Universal Robots PolyScope program: testy.urp

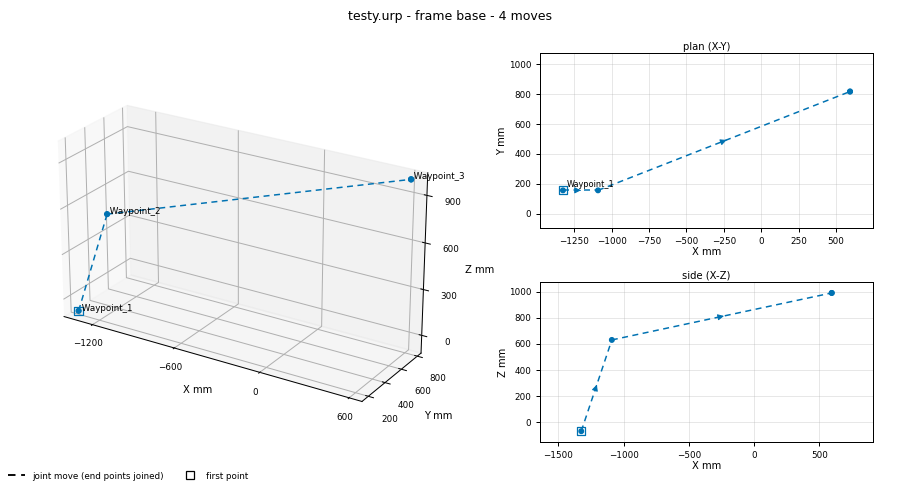
[picture p0: tool path of testy.urp in frame base, 4 of 4 moves have a stored position in this frame; points joined in program order, loops and branches not executed]
Program testy (installation=default directory=/programs createdIn=5.21.3 lastSavedIn=5.21.3 robotSerialNumber=20246801938)
Calibrated DH parameters: a=[-0.000071, -0.790281, -0.600694, 0.000061, -0.000039, 0]; d=[0.236272, 604.465945, 132.116513, -736.382239, 0.159268, 0.154005]; alpha=[1.570254, -0.000567, 0.000559, 1.571709, -1.56999, 0]; deltaTheta=[0, -0.409357, 7.293326, -0.600784, -0.000001, -0.000001]
InitVariablesNode
Robot Program (runOnlyOnce=false)
  'weld angle'
  MoveJ speed 60 deg/s, acceleration 80 deg/s^2 (useActiveTCP=true optimoveEnabled=false optiMoveSpeed=0.3 optiMoveAcceleration=0.09) feature=Base
    Waypoint Waypoint_1: TCP in base x=-1325.071 y=156.59 z=-68.113 mm, rx=-1.7149 ry=0.7798 rz=1.7149 rad; joints [-6.175, -45.066, 109.192, 205.921, -90.048, 42.74] deg; TCP offset x=-11.7 y=-328 z=105 mm, rx=1.2092 ry=-1.2092 rz=1.2092 rad
    Waypoint Waypoint_2: TCP in base x=-1090.841 y=156.59 z=631.078 mm, rx=-1.7149 ry=0.7798 rz=1.7149 rad; joints [-7.848, -90.679, 107.225, 253.5, -89.998, 41.06] deg
  'zero pos'
  MoveJ speed 60 deg/s, acceleration 80 deg/s^2 (useActiveTCP=true optimoveEnabled=false optiMoveSpeed=0.3 optiMoveAcceleration=0.09) feature=Base
    Waypoint Waypoint_3: TCP in base x=593.861 y=817.103 z=991.076 mm, rx=0 ry=0 rz=0 rad; joints [-125.857, -66.581, 112.492, 134.06, -144.207, -0.069] deg
  'first +90 deg y'
  MoveJ speed 60 deg/s, acceleration 80 deg/s^2 (useActiveTCP=true optimoveEnabled=false optiMoveSpeed=0.3 optiMoveAcceleration=0.09) feature=Base
    Waypoint Waypoint_4: TCP in base x=593.863 y=817.112 z=991.08 mm, rx=0 ry=1.5708 rz=0 rad; joints [-121.927, -93.114, 80.917, 282.244, -89.987, 58.062] deg
